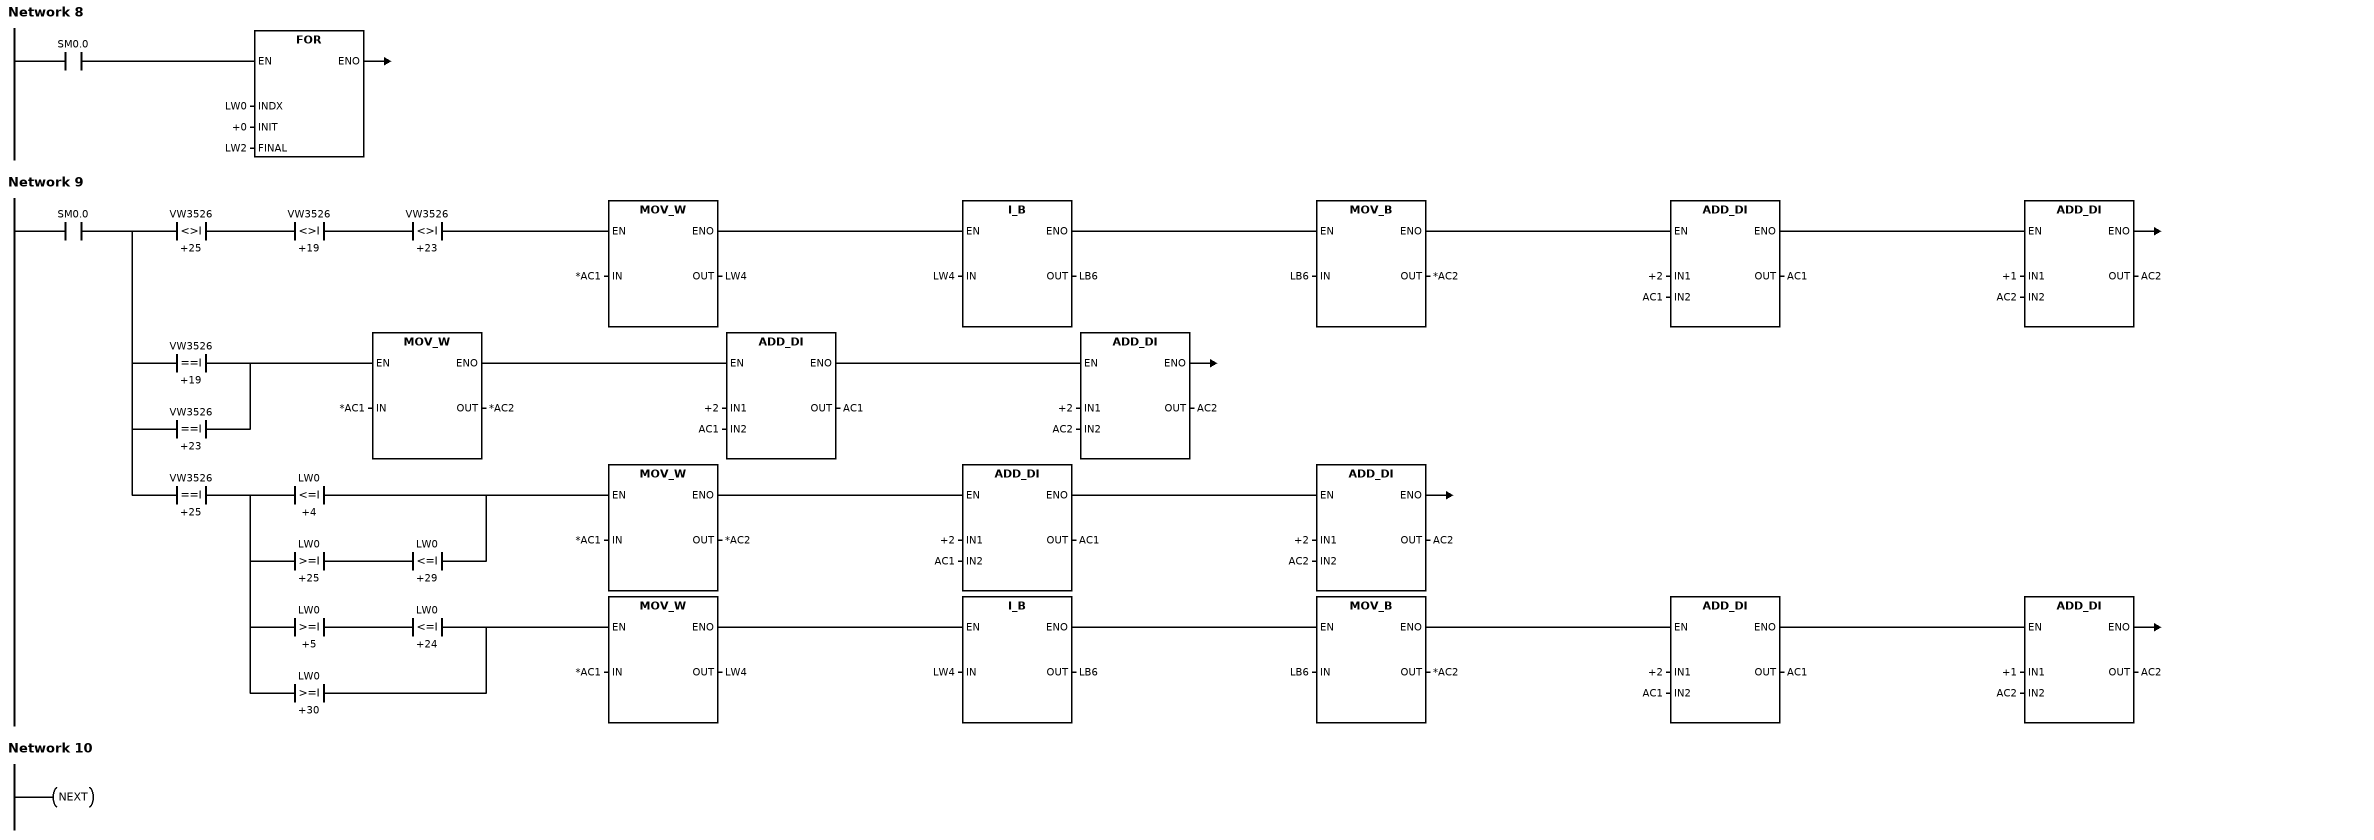
[picture p24: SBR1 networks 8-10]
Network 8
LD     SM0.0
FOR    LW0, +0, LW2
Network 9
LD     SM0.0
LPS
AW<>   VW3526, +25
AW<>   VW3526, +19
AW<>   VW3526, +23
MOVW   *AC1, LW4
AENO
ITB    LW4, LB6
AENO
MOVB   LB6, *AC2
AENO
+D     +2, AC1
AENO
+D     +1, AC2
LRD
LDW=   VW3526, +19
OW=    VW3526, +23
ALD
MOVW   *AC1, *AC2
AENO
+D     +2, AC1
AENO
+D     +2, AC2
LPP
AW=    VW3526, +25
LPS
LDW<=  LW0, +4
LDW>=  LW0, +25
AW<=   LW0, +29
OLD
ALD
MOVW   *AC1, *AC2
AENO
+D     +2, AC1
AENO
+D     +2, AC2
LPP
LDW>=  LW0, +5
AW<=   LW0, +24
OW>=   LW0, +30
ALD
MOVW   *AC1, LW4
AENO
ITB    LW4, LB6
AENO
MOVB   LB6, *AC2
AENO
+D     +2, AC1
AENO
+D     +1, AC2
Network 10
NEXT
END_SUBROUTINE_BLOCK

SUBROUTINE_BLOCK STATION_ZK:SBR2
TITLE=
BEGIN
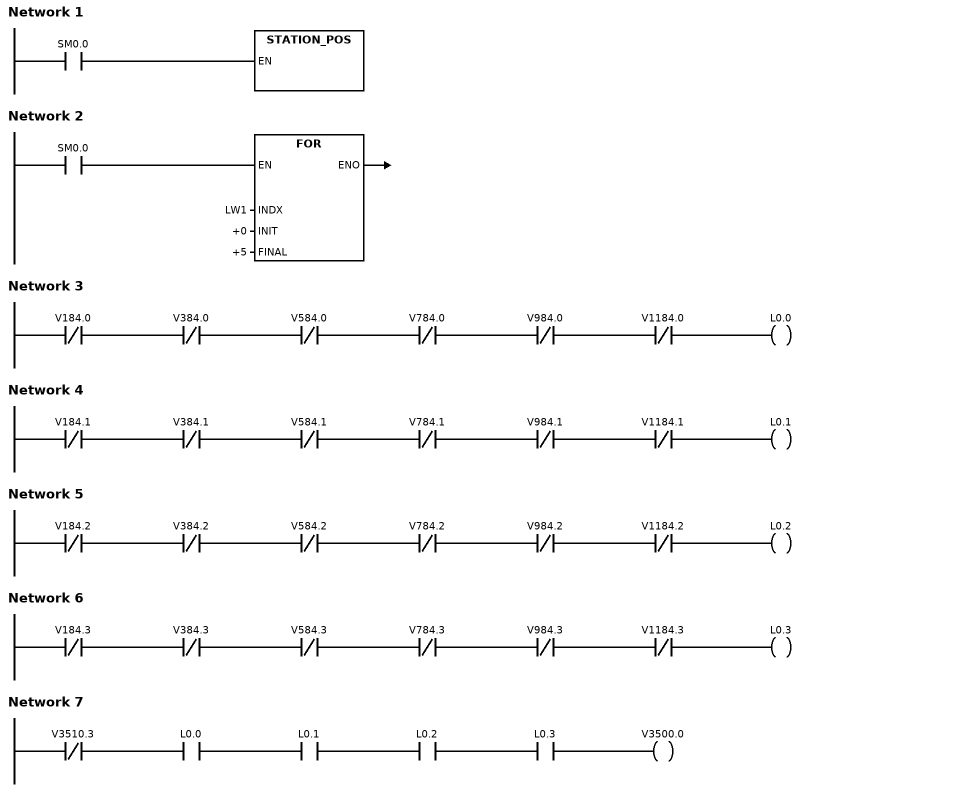
Network 1
LD     SM0.0
CALL   STATION_POS:SBR7
Network 2
LD     SM0.0
FOR    LW1, +0, +5
Network 3
LDN    V184.0
AN     V384.0
AN     V584.0
AN     V784.0
AN     V984.0
AN     V1184.0
=      L0.0
Network 4
LDN    V184.1
AN     V384.1
AN     V584.1
AN     V784.1
AN     V984.1
AN     V1184.1
=      L0.1
Network 5
LDN    V184.2
AN     V384.2
AN     V584.2
AN     V784.2
AN     V984.2
AN     V1184.2
=      L0.2
Network 6
LDN    V184.3
AN     V384.3
AN     V584.3
AN     V784.3
AN     V984.3
AN     V1184.3
=      L0.3
Network 7
LDN    V3510.3
A      L0.0
A      L0.1
A      L0.2
A      L0.3
=      V3500.0
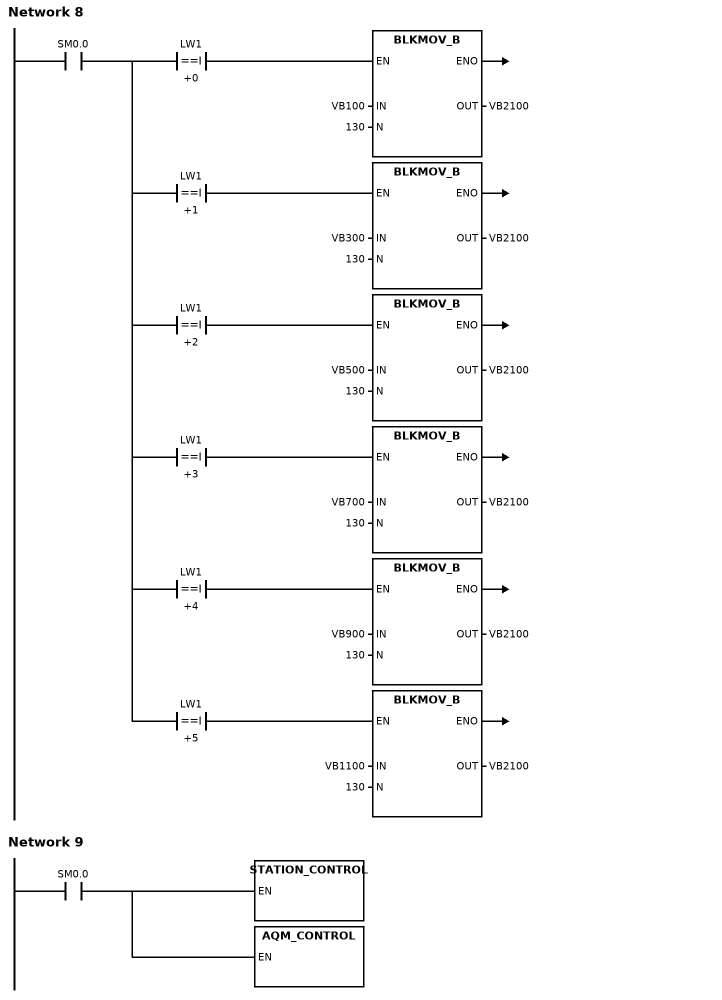
Network 8
LD     SM0.0
LPS
AW=    LW1, +0
BMB    VB100, VB2100, 130
LRD
AW=    LW1, +1
BMB    VB300, VB2100, 130
LRD
AW=    LW1, +2
BMB    VB500, VB2100, 130
LRD
AW=    LW1, +3
BMB    VB700, VB2100, 130
LRD
AW=    LW1, +4
BMB    VB900, VB2100, 130
LPP
AW=    LW1, +5
BMB    VB1100, VB2100, 130
Network 9
LD     SM0.0
CALL   STATION_CONTROL:SBR0
CALL   AQM_CONTROL:SBR8
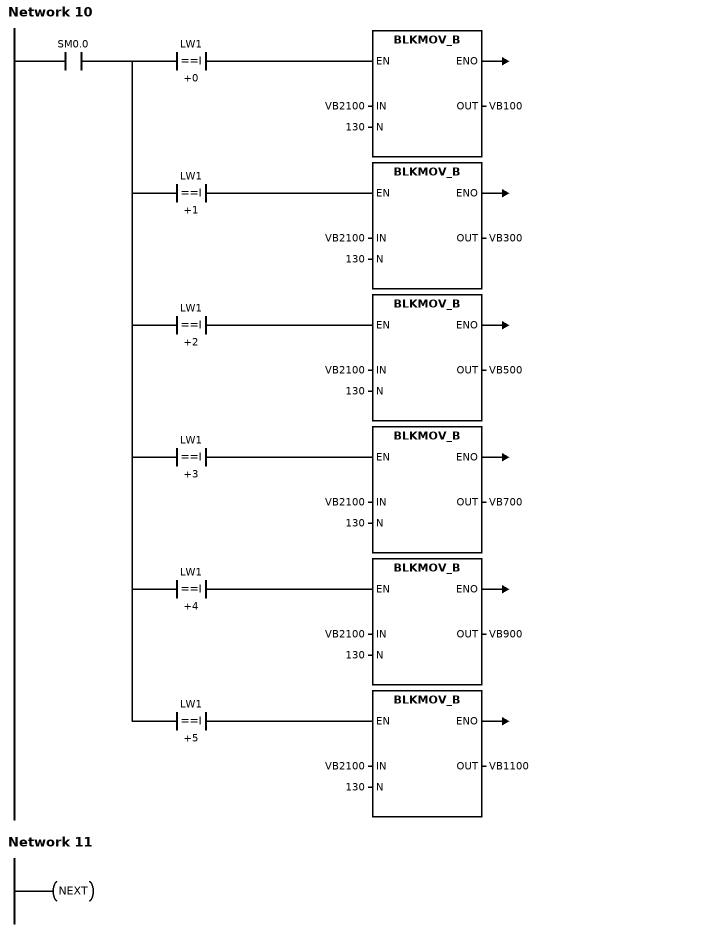
Network 10
LD     SM0.0
LPS
AW=    LW1, +0
BMB    VB2100, VB100, 130
LRD
AW=    LW1, +1
BMB    VB2100, VB300, 130
LRD
AW=    LW1, +2
BMB    VB2100, VB500, 130
LRD
AW=    LW1, +3
BMB    VB2100, VB700, 130
LRD
AW=    LW1, +4
BMB    VB2100, VB900, 130
LPP
AW=    LW1, +5
BMB    VB2100, VB1100, 130
Network 11
NEXT
END_SUBROUTINE_BLOCK

SUBROUTINE_BLOCK YX_YLKZ:SBR3
TITLE=
BEGIN
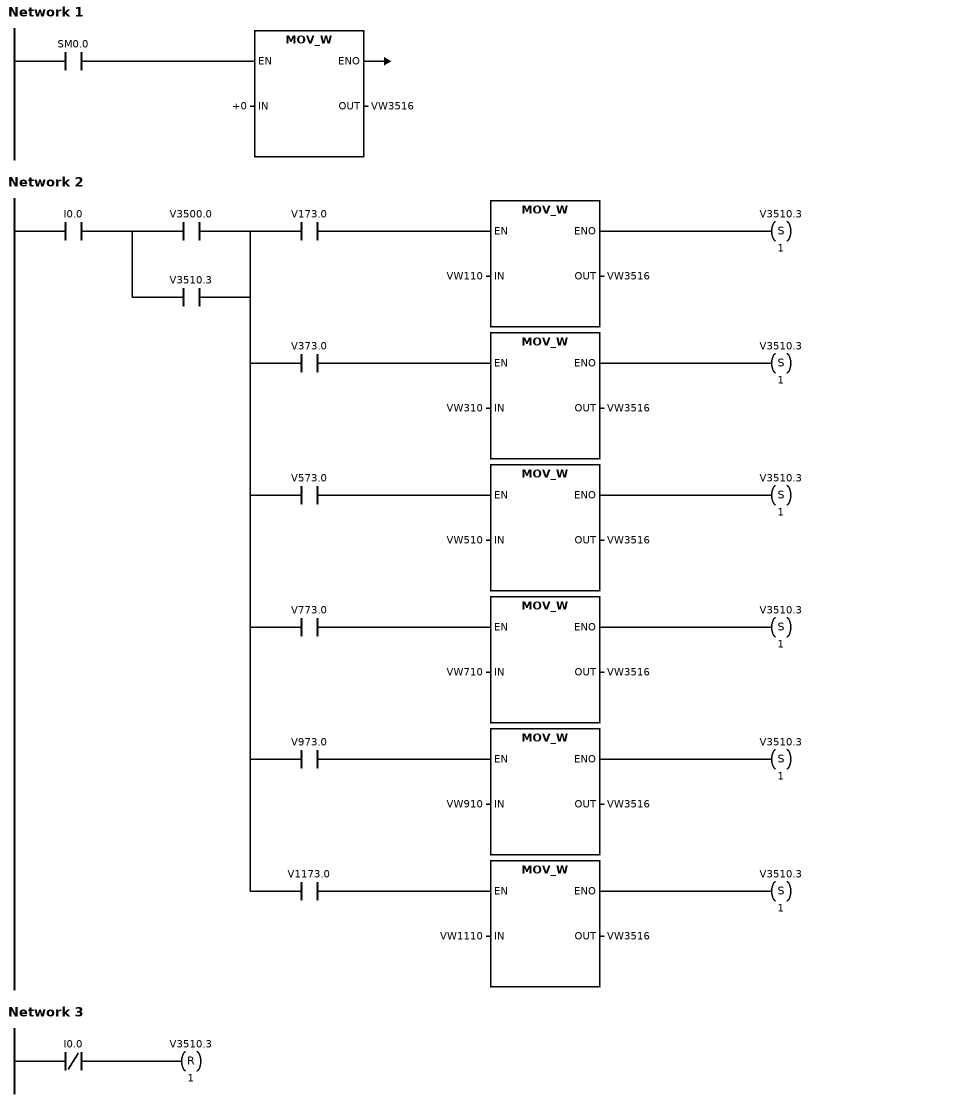
Network 1
LD     SM0.0
MOVW   +0, VW3516
Network 2
LD     I0.0
LD     V3500.0
O      V3510.3
ALD
LPS
A      V173.0
MOVW   VW110, VW3516
AENO
S      V3510.3, 1
LRD
A      V373.0
MOVW   VW310, VW3516
AENO
S      V3510.3, 1
LRD
A      V573.0
MOVW   VW510, VW3516
AENO
S      V3510.3, 1
LRD
A      V773.0
MOVW   VW710, VW3516
AENO
S      V3510.3, 1
LRD
A      V973.0
MOVW   VW910, VW3516
AENO
S      V3510.3, 1
LPP
A      V1173.0
MOVW   VW1110, VW3516
AENO
S      V3510.3, 1
Network 3
LDN    I0.0
R      V3510.3, 1
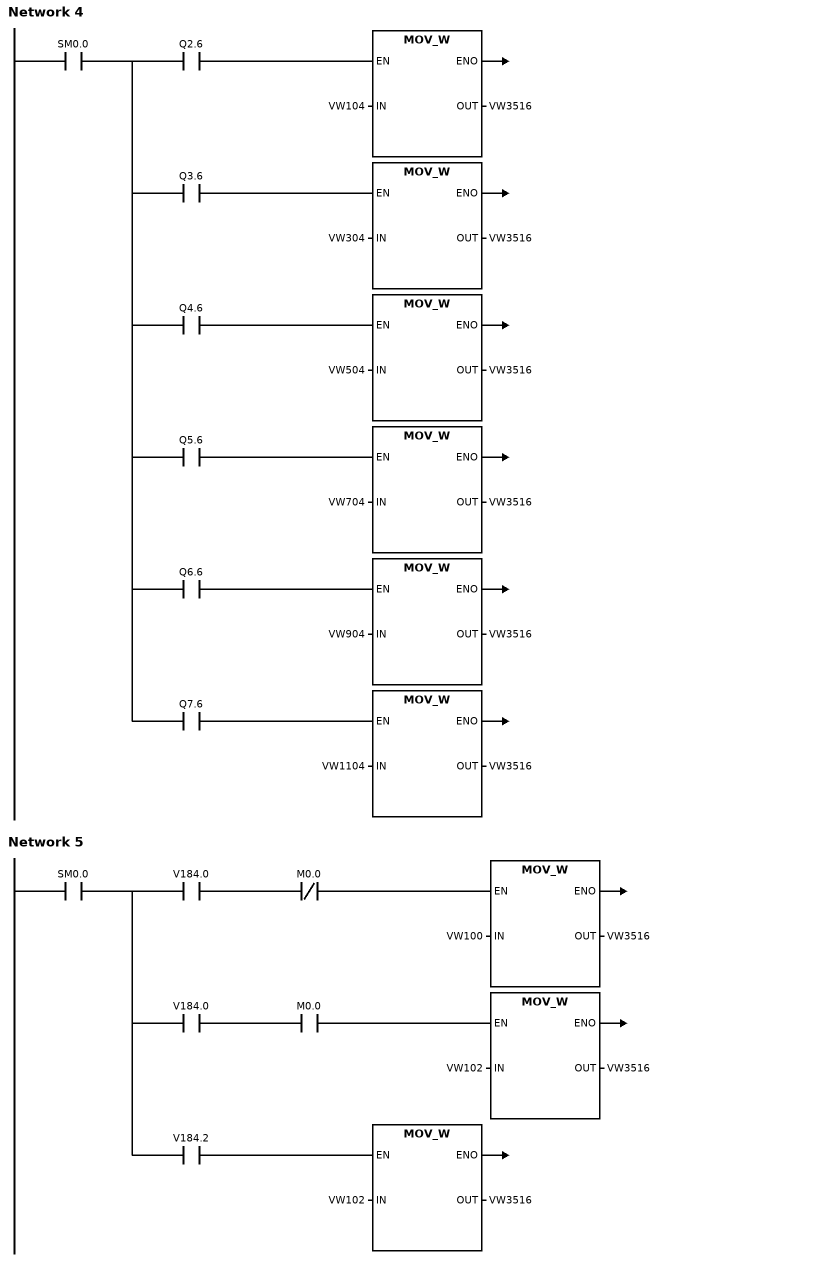
Network 4
LD     SM0.0
LPS
A      Q2.6
MOVW   VW104, VW3516
LRD
A      Q3.6
MOVW   VW304, VW3516
LRD
A      Q4.6
MOVW   VW504, VW3516
LRD
A      Q5.6
MOVW   VW704, VW3516
LRD
A      Q6.6
MOVW   VW904, VW3516
LPP
A      Q7.6
MOVW   VW1104, VW3516
Network 5
LD     SM0.0
LPS
A      V184.0
AN     M0.0
MOVW   VW100, VW3516
LRD
A      V184.0
A      M0.0
MOVW   VW102, VW3516
LPP
A      V184.2
MOVW   VW102, VW3516
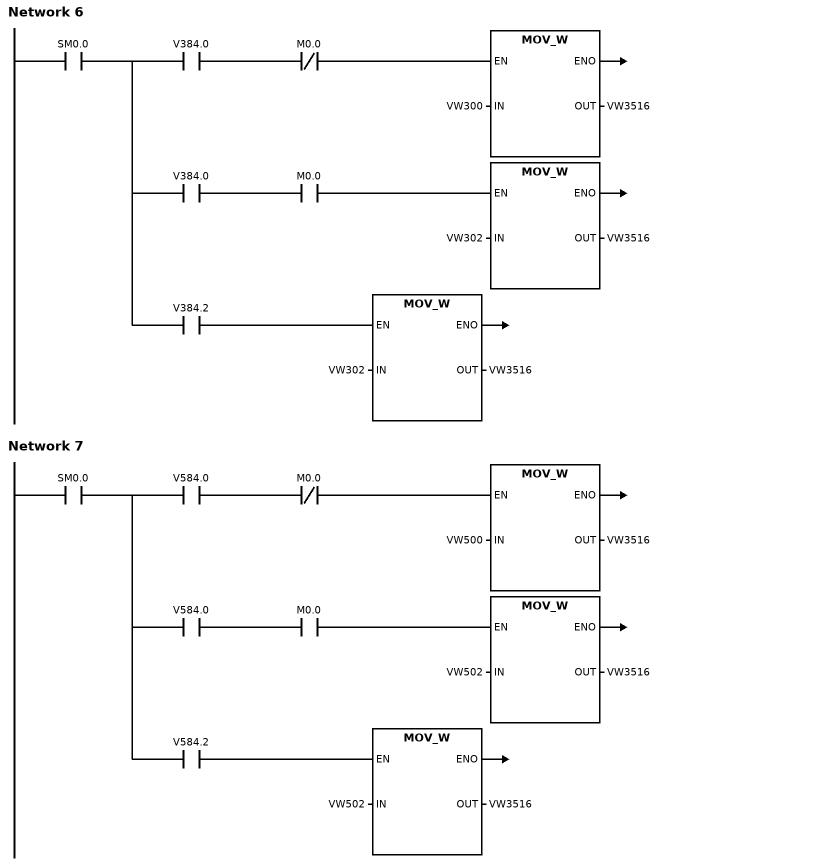
Network 6
LD     SM0.0
LPS
A      V384.0
AN     M0.0
MOVW   VW300, VW3516
LRD
A      V384.0
A      M0.0
MOVW   VW302, VW3516
LPP
A      V384.2
MOVW   VW302, VW3516
Network 7
LD     SM0.0
LPS
A      V584.0
AN     M0.0
MOVW   VW500, VW3516
LRD
A      V584.0
A      M0.0
MOVW   VW502, VW3516
LPP
A      V584.2
MOVW   VW502, VW3516
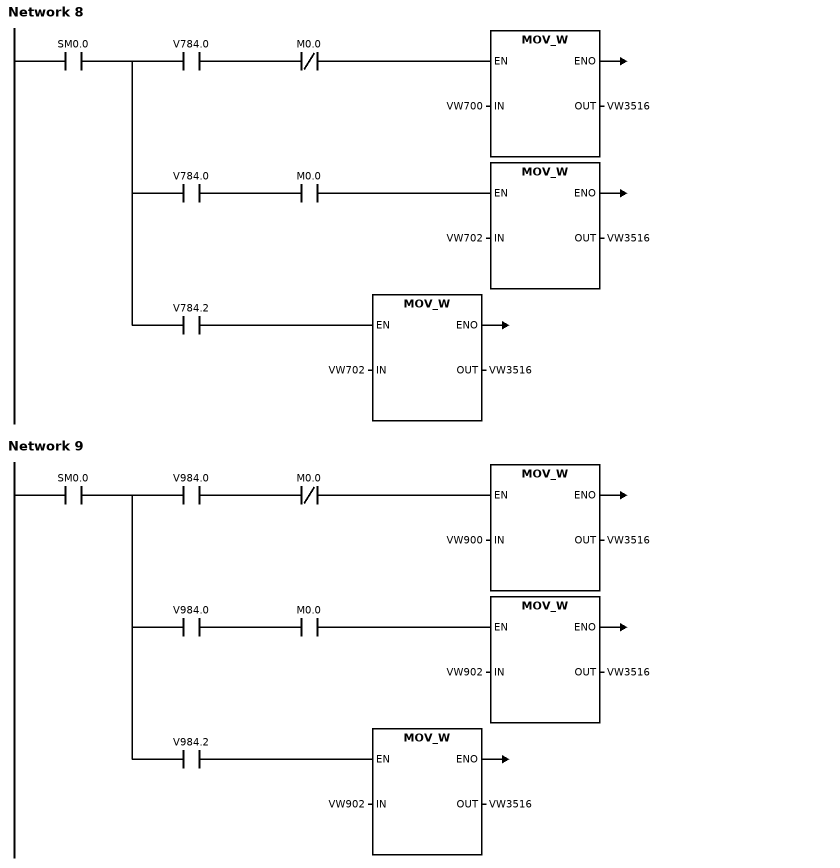
Network 8
LD     SM0.0
LPS
A      V784.0
AN     M0.0
MOVW   VW700, VW3516
LRD
A      V784.0
A      M0.0
MOVW   VW702, VW3516
LPP
A      V784.2
MOVW   VW702, VW3516
Network 9
LD     SM0.0
LPS
A      V984.0
AN     M0.0
MOVW   VW900, VW3516
LRD
A      V984.0
A      M0.0
MOVW   VW902, VW3516
LPP
A      V984.2
MOVW   VW902, VW3516
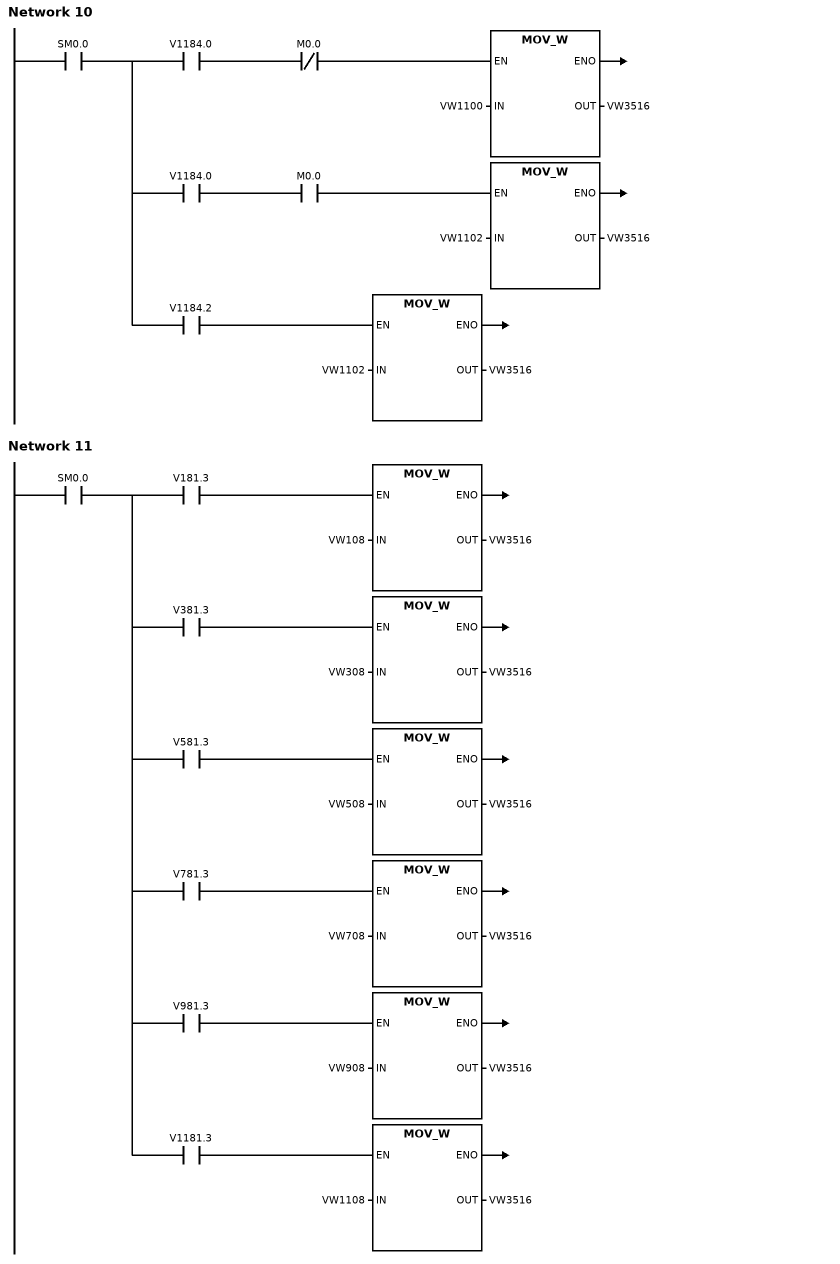
Network 10
LD     SM0.0
LPS
A      V1184.0
AN     M0.0
MOVW   VW1100, VW3516
LRD
A      V1184.0
A      M0.0
MOVW   VW1102, VW3516
LPP
A      V1184.2
MOVW   VW1102, VW3516
Network 11
LD     SM0.0
LPS
A      V181.3
MOVW   VW108, VW3516
LRD
A      V381.3
MOVW   VW308, VW3516
LRD
A      V581.3
MOVW   VW508, VW3516
LRD
A      V781.3
MOVW   VW708, VW3516
LRD
A      V981.3
MOVW   VW908, VW3516
LPP
A      V1181.3
MOVW   VW1108, VW3516
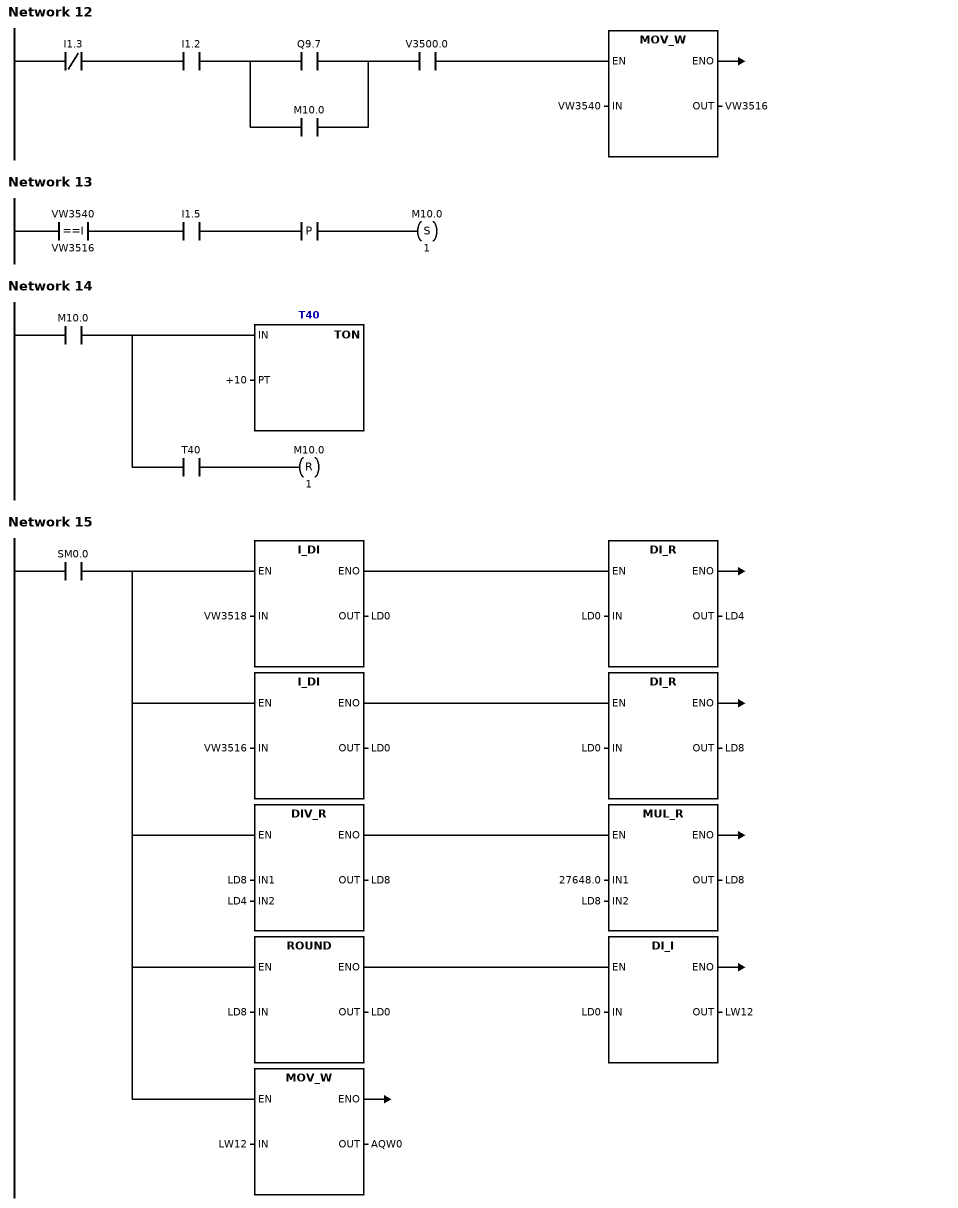
Network 12
LDN    I1.3
A      I1.2
LD     Q9.7
O      M10.0
ALD
A      V3500.0
MOVW   VW3540, VW3516
Network 13
LDW=   VW3540, VW3516
A      I1.5
EU
S      M10.0, 1
Network 14
LD     M10.0
TON    T40, +10
A      T40
R      M10.0, 1
Network 15
LD     SM0.0
LPS
ITD    VW3518, LD0
AENO
DTR    LD0, LD4
LRD
ITD    VW3516, LD0
AENO
DTR    LD0, LD8
LRD
/R     LD4, LD8
AENO
*R     27648.0, LD8
LRD
ROUND  LD8, LD0
AENO
DTI    LD0, LW12
LPP
MOVW   LW12, AQW0
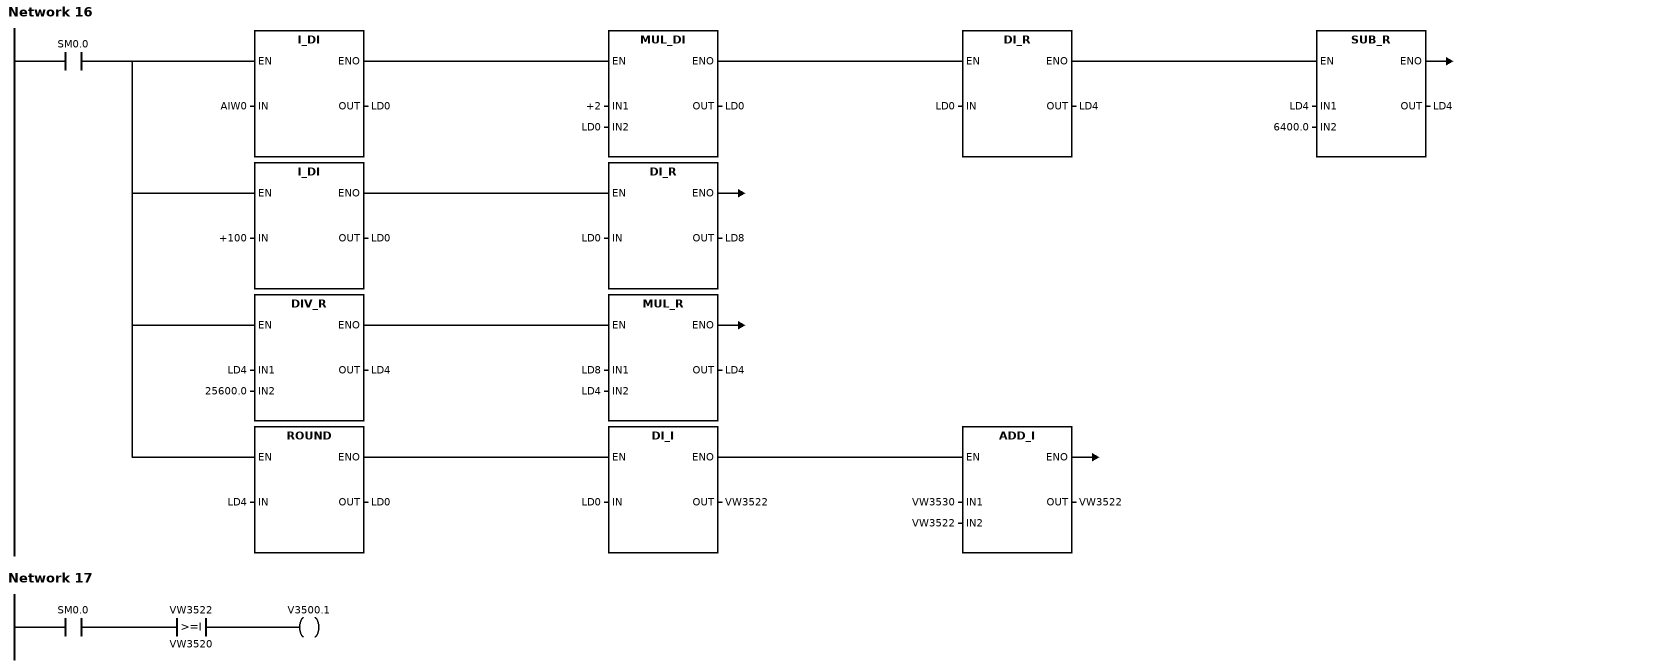
Network 16
LD     SM0.0
LPS
ITD    AIW0, LD0
AENO
*D     +2, LD0
AENO
DTR    LD0, LD4
AENO
-R     6400.0, LD4
LRD
ITD    +100, LD0
AENO
DTR    LD0, LD8
LRD
/R     25600.0, LD4
AENO
*R     LD8, LD4
LPP
ROUND  LD4, LD0
AENO
DTI    LD0, VW3522
AENO
+I     VW3530, VW3522
Network 17
LD     SM0.0
AW>=   VW3522, VW3520
=      V3500.1
END_SUBROUTINE_BLOCK

SUBROUTINE_BLOCK DI_EXCHANGE:SBR4
TITLE=
BEGIN
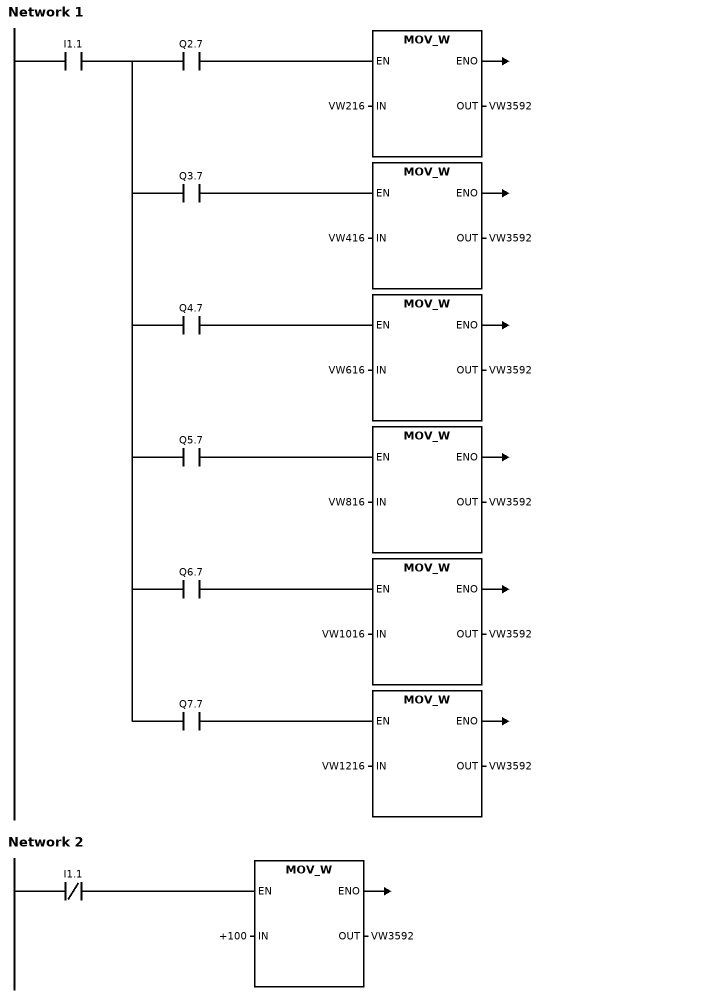
Network 1
LD     I1.1
LPS
A      Q2.7
MOVW   VW216, VW3592
LRD
A      Q3.7
MOVW   VW416, VW3592
LRD
A      Q4.7
MOVW   VW616, VW3592
LRD
A      Q5.7
MOVW   VW816, VW3592
LRD
A      Q6.7
MOVW   VW1016, VW3592
LPP
A      Q7.7
MOVW   VW1216, VW3592
Network 2
LDN    I1.1
MOVW   +100, VW3592
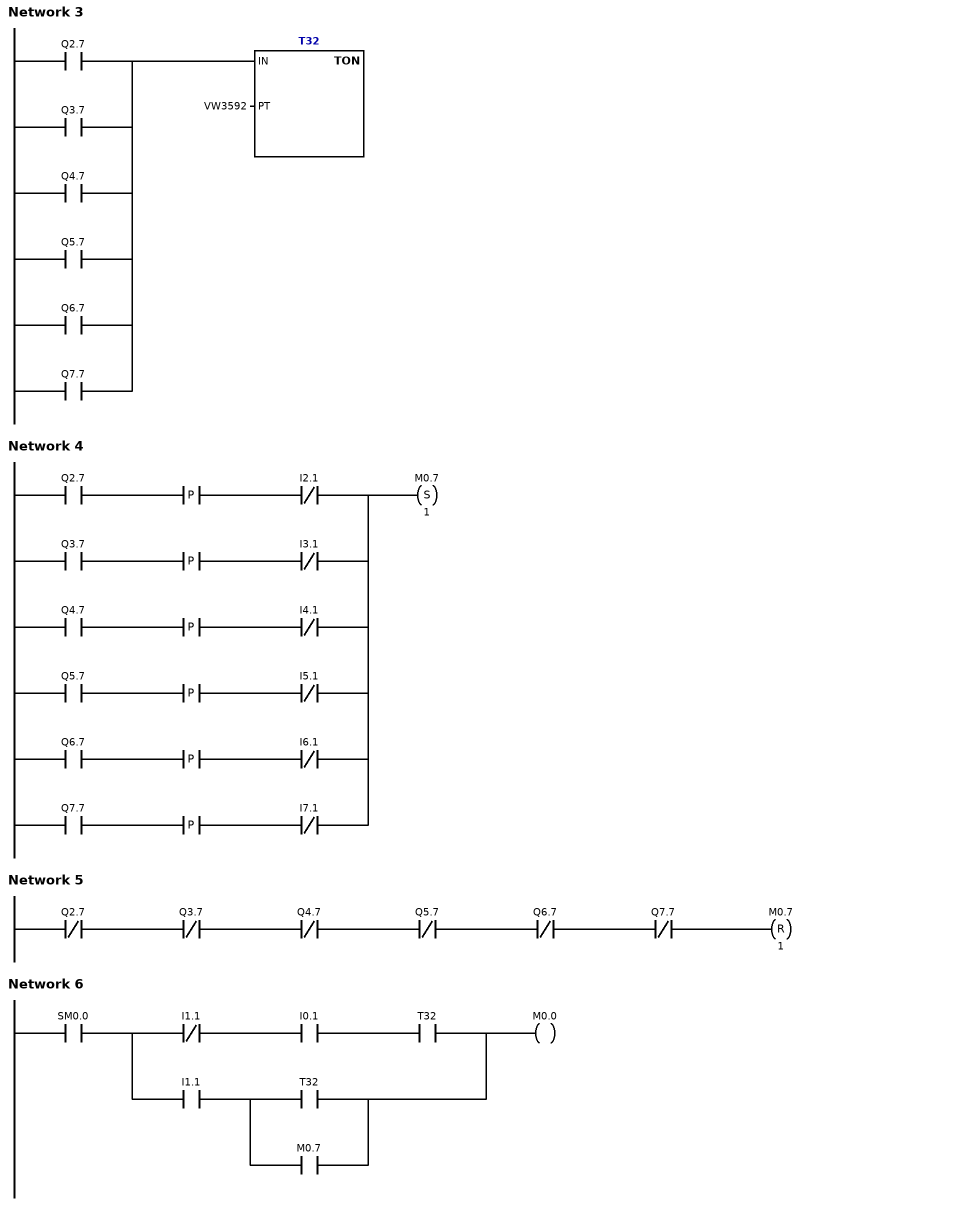
Network 3
LD     Q2.7
O      Q3.7
O      Q4.7
O      Q5.7
O      Q6.7
O      Q7.7
TON    T32, VW3592
Network 4
LD     Q2.7
EU
AN     I2.1
LD     Q3.7
EU
AN     I3.1
OLD
LD     Q4.7
EU
AN     I4.1
OLD
LD     Q5.7
EU
AN     I5.1
OLD
LD     Q6.7
EU
AN     I6.1
OLD
LD     Q7.7
EU
AN     I7.1
OLD
S      M0.7, 1
Network 5
LDN    Q2.7
AN     Q3.7
AN     Q4.7
AN     Q5.7
AN     Q6.7
AN     Q7.7
R      M0.7, 1
Network 6
LD     SM0.0
LDN    I1.1
A      I0.1
A      T32
LD     I1.1
LD     T32
O      M0.7
ALD
OLD
ALD
=      M0.0
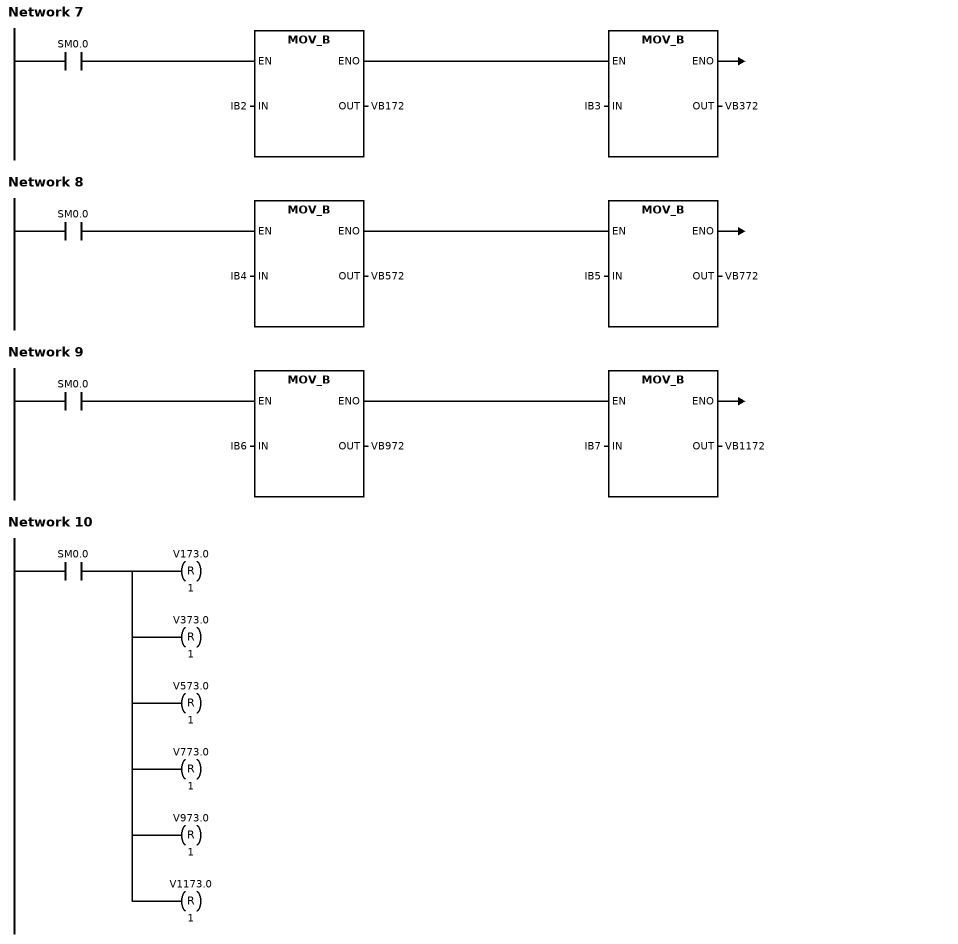
Network 7
LD     SM0.0
MOVB   IB2, VB172
AENO
MOVB   IB3, VB372
Network 8
LD     SM0.0
MOVB   IB4, VB572
AENO
MOVB   IB5, VB772
Network 9
LD     SM0.0
MOVB   IB6, VB972
AENO
MOVB   IB7, VB1172
Network 10
LD     SM0.0
R      V173.0, 1
R      V373.0, 1
R      V573.0, 1
R      V773.0, 1
R      V973.0, 1
R      V1173.0, 1
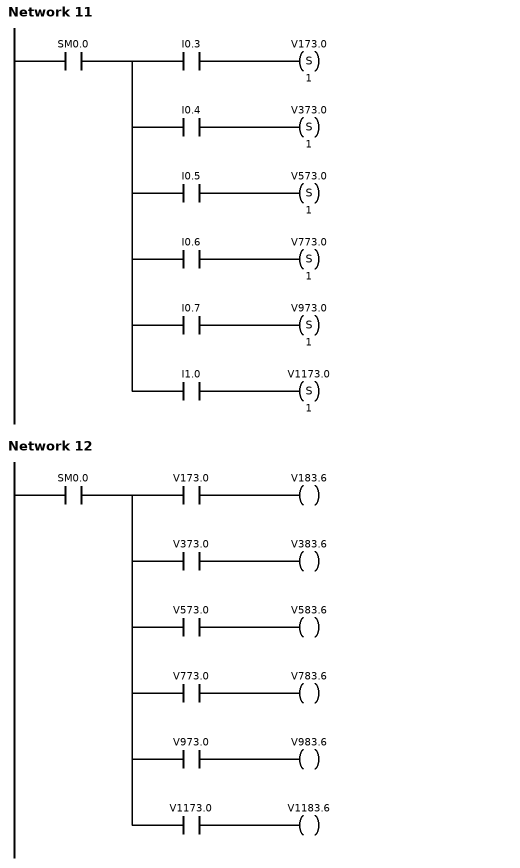
Network 11
LD     SM0.0
LPS
A      I0.3
S      V173.0, 1
LRD
A      I0.4
S      V373.0, 1
LRD
A      I0.5
S      V573.0, 1
LRD
A      I0.6
S      V773.0, 1
LRD
A      I0.7
S      V973.0, 1
LPP
A      I1.0
S      V1173.0, 1
Network 12
LD     SM0.0
LPS
A      V173.0
=      V183.6
LRD
A      V373.0
=      V383.6
LRD
A      V573.0
=      V583.6
LRD
A      V773.0
=      V783.6
LRD
A      V973.0
=      V983.6
LPP
A      V1173.0
=      V1183.6
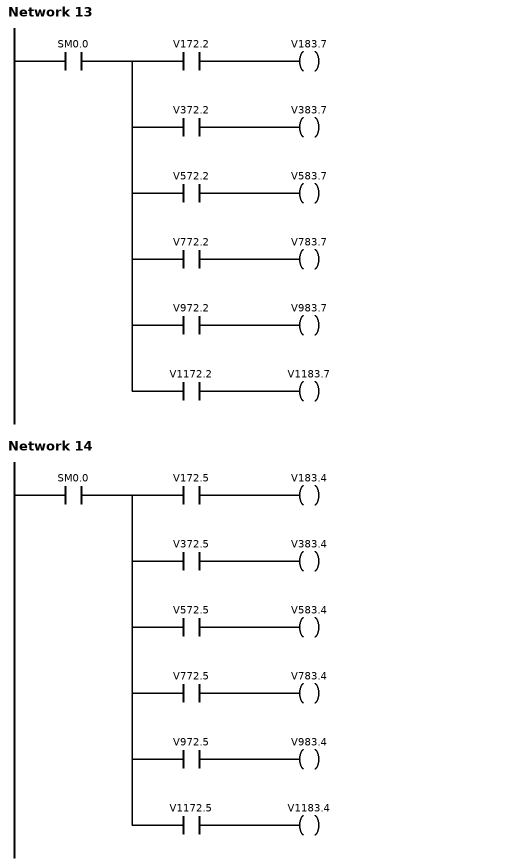
Network 13
LD     SM0.0
LPS
A      V172.2
=      V183.7
LRD
A      V372.2
=      V383.7
LRD
A      V572.2
=      V583.7
LRD
A      V772.2
=      V783.7
LRD
A      V972.2
=      V983.7
LPP
A      V1172.2
=      V1183.7
Network 14
LD     SM0.0
LPS
A      V172.5
=      V183.4
LRD
A      V372.5
=      V383.4
LRD
A      V572.5
=      V583.4
LRD
A      V772.5
=      V783.4
LRD
A      V972.5
=      V983.4
LPP
A      V1172.5
=      V1183.4
END_SUBROUTINE_BLOCK

SUBROUTINE_BLOCK DO_EXCHANGE:SBR5
TITLE=
BEGIN
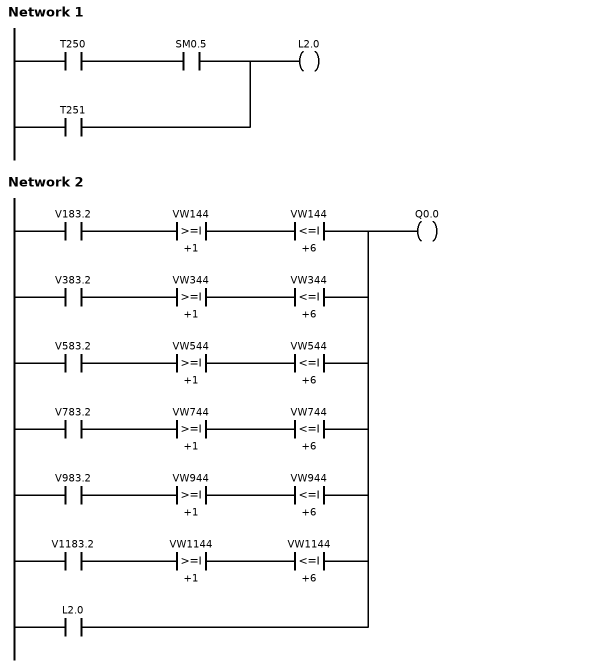
Network 1
LD     T250
A      SM0.5
O      T251
=      L2.0
Network 2
LD     V183.2
AW>=   VW144, +1
AW<=   VW144, +6
LD     V383.2
AW>=   VW344, +1
AW<=   VW344, +6
OLD
LD     V583.2
AW>=   VW544, +1
AW<=   VW544, +6
OLD
LD     V783.2
AW>=   VW744, +1
AW<=   VW744, +6
OLD
LD     V983.2
AW>=   VW944, +1
AW<=   VW944, +6
OLD
LD     V1183.2
AW>=   VW1144, +1
AW<=   VW1144, +6
OLD
O      L2.0
=      Q0.0
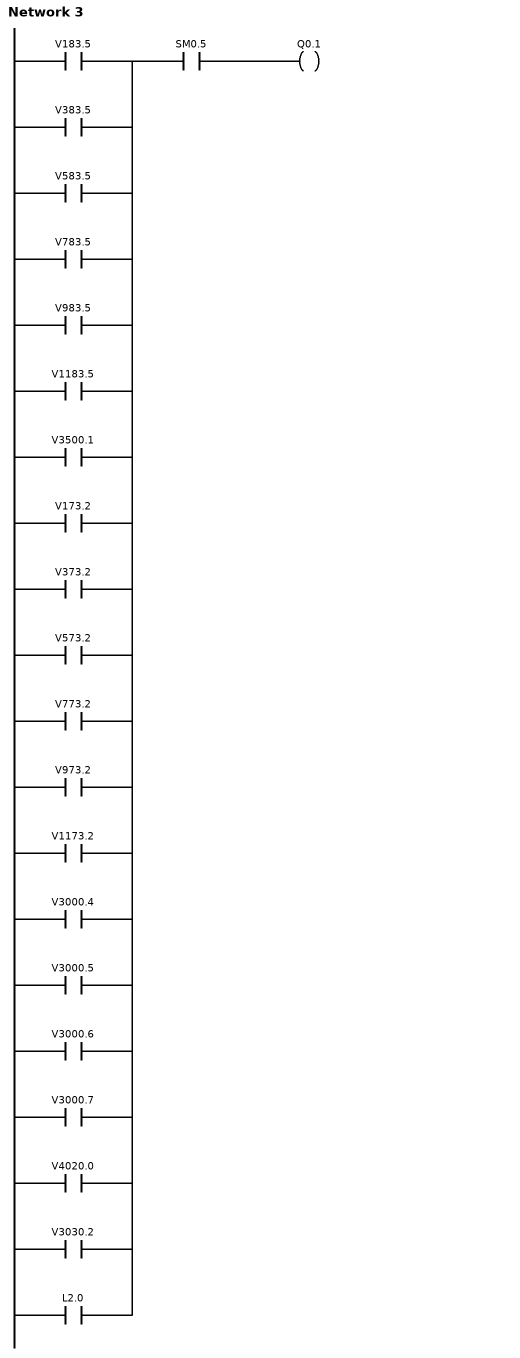
Network 3
LD     V183.5
O      V383.5
O      V583.5
O      V783.5
O      V983.5
O      V1183.5
O      V3500.1
O      V173.2
O      V373.2
O      V573.2
O      V773.2
O      V973.2
O      V1173.2
O      V3000.4
O      V3000.5
O      V3000.6
O      V3000.7
O      V4020.0
O      V3030.2
O      L2.0
A      SM0.5
=      Q0.1
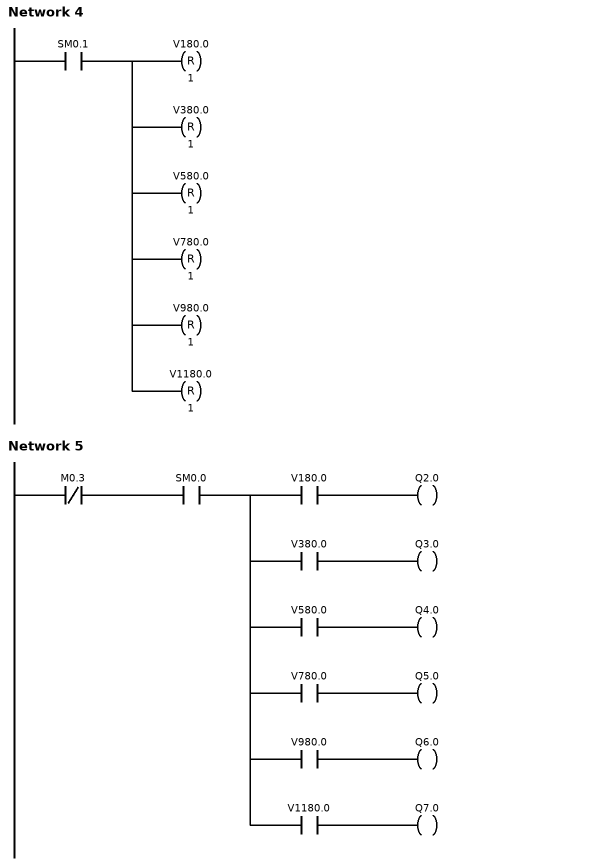
Network 4
LD     SM0.1
R      V180.0, 1
R      V380.0, 1
R      V580.0, 1
R      V780.0, 1
R      V980.0, 1
R      V1180.0, 1
Network 5
LDN    M0.3
A      SM0.0
LPS
A      V180.0
=      Q2.0
LRD
A      V380.0
=      Q3.0
LRD
A      V580.0
=      Q4.0
LRD
A      V780.0
=      Q5.0
LRD
A      V980.0
=      Q6.0
LPP
A      V1180.0
=      Q7.0
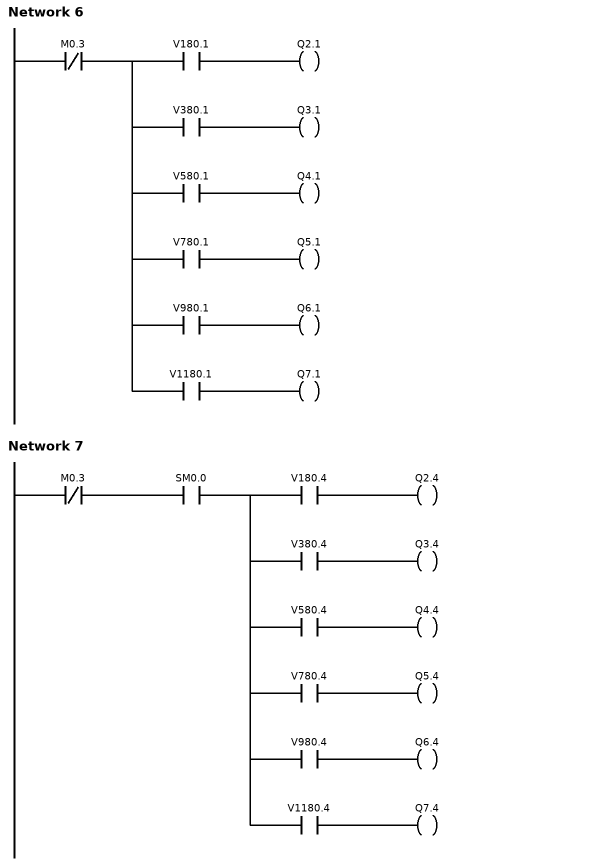
Network 6
LDN    M0.3
LPS
A      V180.1
=      Q2.1
LRD
A      V380.1
=      Q3.1
LRD
A      V580.1
=      Q4.1
LRD
A      V780.1
=      Q5.1
LRD
A      V980.1
=      Q6.1
LPP
A      V1180.1
=      Q7.1
Network 7
LDN    M0.3
A      SM0.0
LPS
A      V180.4
=      Q2.4
LRD
A      V380.4
=      Q3.4
LRD
A      V580.4
=      Q4.4
LRD
A      V780.4
=      Q5.4
LRD
A      V980.4
=      Q6.4
LPP
A      V1180.4
=      Q7.4
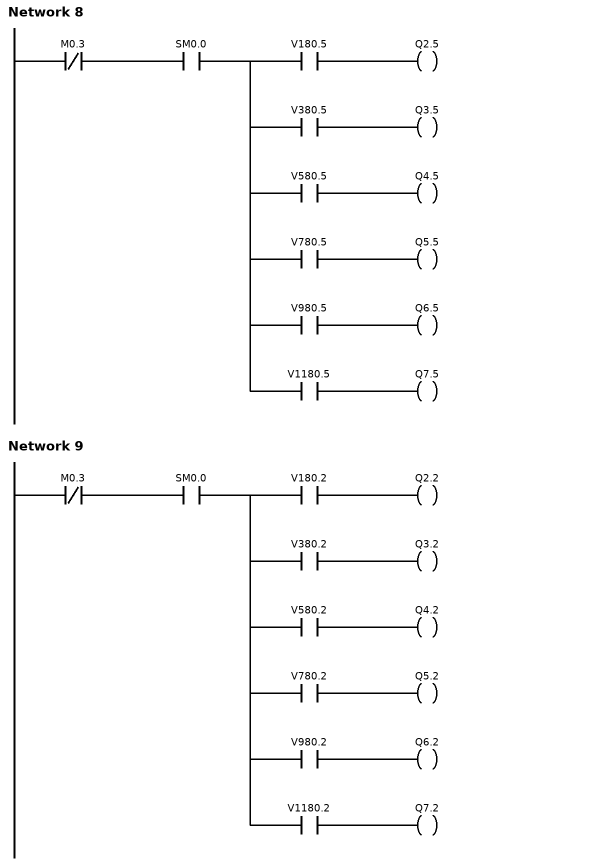
Network 8
LDN    M0.3
A      SM0.0
LPS
A      V180.5
=      Q2.5
LRD
A      V380.5
=      Q3.5
LRD
A      V580.5
=      Q4.5
LRD
A      V780.5
=      Q5.5
LRD
A      V980.5
=      Q6.5
LPP
A      V1180.5
=      Q7.5
Network 9
LDN    M0.3
A      SM0.0
LPS
A      V180.2
=      Q2.2
LRD
A      V380.2
=      Q3.2
LRD
A      V580.2
=      Q4.2
LRD
A      V780.2
=      Q5.2
LRD
A      V980.2
=      Q6.2
LPP
A      V1180.2
=      Q7.2
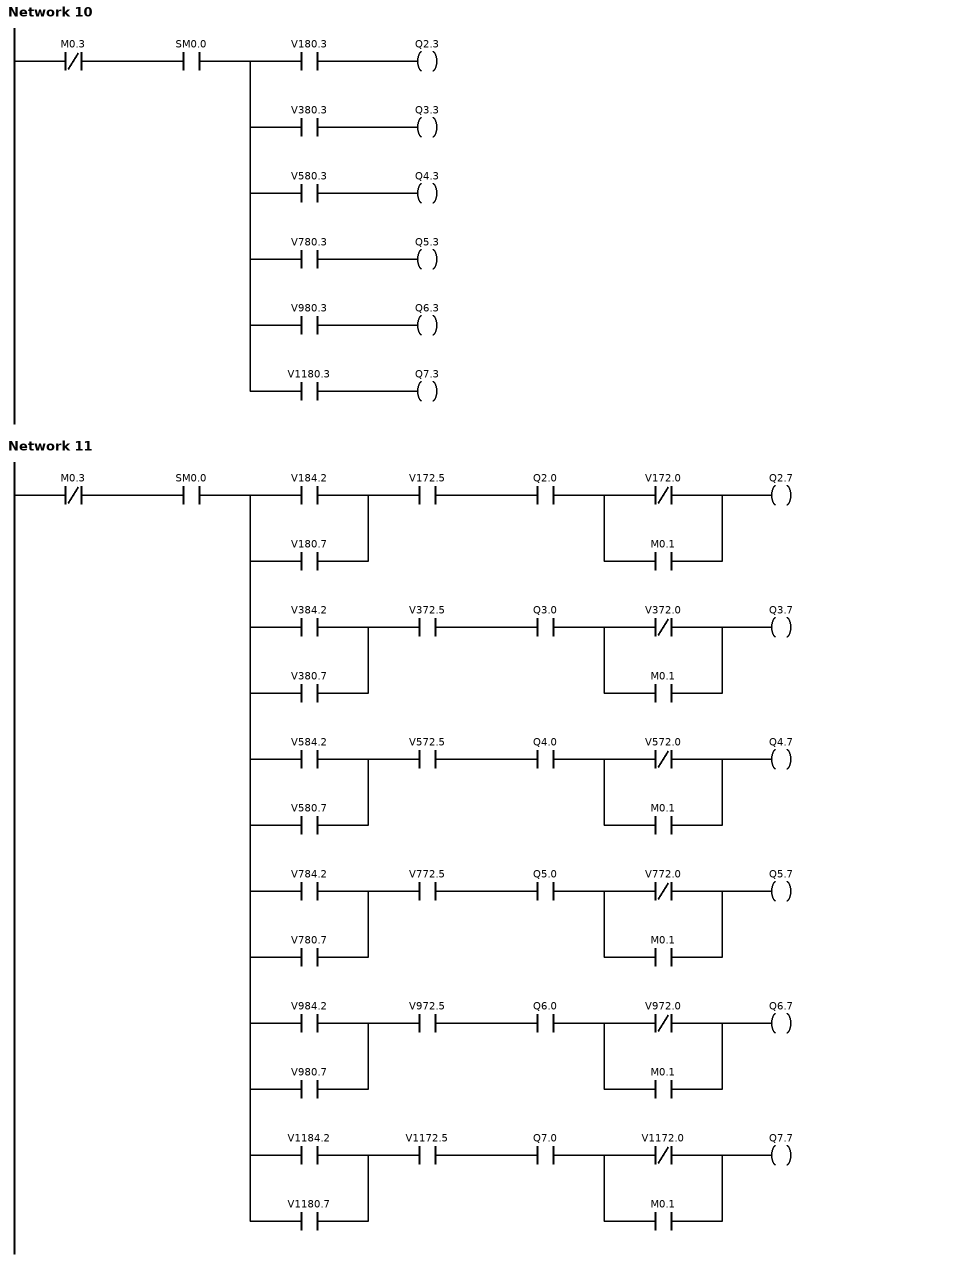
Network 10
LDN    M0.3
A      SM0.0
LPS
A      V180.3
=      Q2.3
LRD
A      V380.3
=      Q3.3
LRD
A      V580.3
=      Q4.3
LRD
A      V780.3
=      Q5.3
LRD
A      V980.3
=      Q6.3
LPP
A      V1180.3
=      Q7.3
Network 11
LDN    M0.3
A      SM0.0
LPS
LD     V184.2
O      V180.7
A      V172.5
A      Q2.0
LDN    V172.0
O      M0.1
ALD
ALD
=      Q2.7
LRD
LD     V384.2
O      V380.7
A      V372.5
A      Q3.0
LDN    V372.0
O      M0.1
ALD
ALD
=      Q3.7
LRD
LD     V584.2
O      V580.7
A      V572.5
A      Q4.0
LDN    V572.0
O      M0.1
ALD
ALD
=      Q4.7
LRD
LD     V784.2
O      V780.7
A      V772.5
A      Q5.0
LDN    V772.0
O      M0.1
ALD
ALD
=      Q5.7
LRD
LD     V984.2
O      V980.7
A      V972.5
A      Q6.0
LDN    V972.0
O      M0.1
ALD
ALD
=      Q6.7
LPP
LD     V1184.2
O      V1180.7
A      V1172.5
A      Q7.0
LDN    V1172.0
O      M0.1
ALD
ALD
=      Q7.7
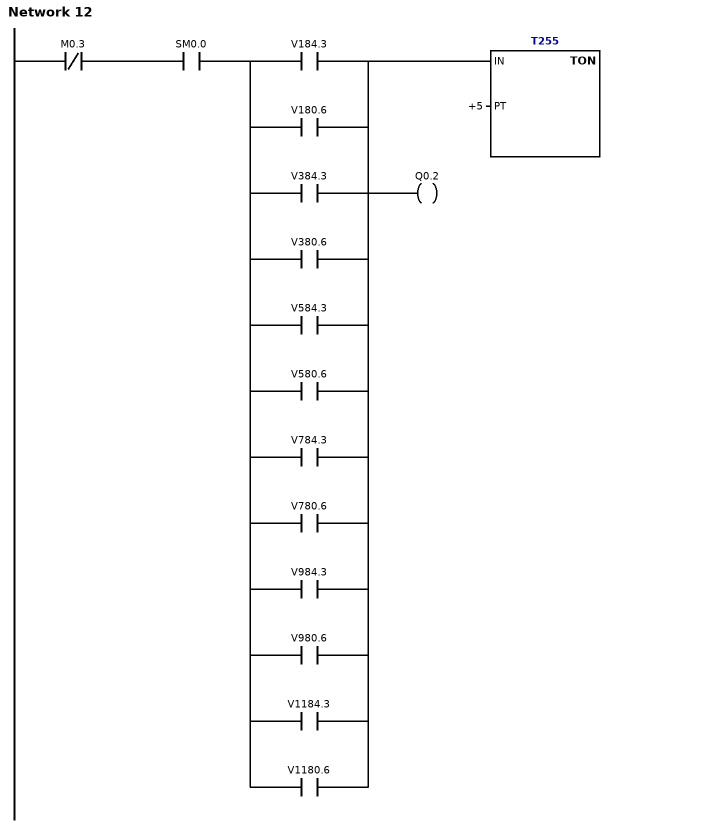
Network 12
LDN    M0.3
A      SM0.0
LD     V184.3
O      V180.6
O      V384.3
O      V380.6
O      V584.3
O      V580.6
O      V784.3
O      V780.6
O      V984.3
O      V980.6
O      V1184.3
O      V1180.6
ALD
TON    T255, +5
=      Q0.2
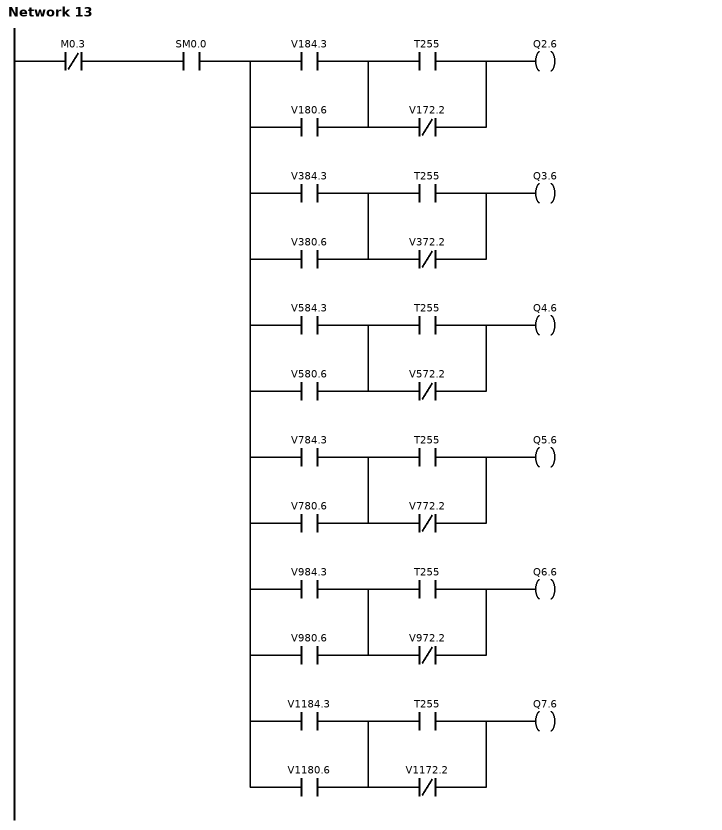
Network 13
LDN    M0.3
A      SM0.0
LPS
LD     V184.3
O      V180.6
LD     T255
ON     V172.2
ALD
ALD
=      Q2.6
LRD
LD     V384.3
O      V380.6
LD     T255
ON     V372.2
ALD
ALD
=      Q3.6
LRD
LD     V584.3
O      V580.6
LD     T255
ON     V572.2
ALD
ALD
=      Q4.6
LRD
LD     V784.3
O      V780.6
LD     T255
ON     V772.2
ALD
ALD
=      Q5.6
LRD
LD     V984.3
O      V980.6
LD     T255
ON     V972.2
ALD
ALD
=      Q6.6
LPP
LD     V1184.3
O      V1180.6
LD     T255
ON     V1172.2
ALD
ALD
=      Q7.6
